//---------------------------------------------------------------------------------------------------------------
//
//  HAUD 2025.08.20
//
//  - XTS_TRANSPORT_LAYER
//
//  fb_StationBase
//  - abstract base class for XtsStation and XtsStationGearIn to extend
//  - anything goes..
//    - if you need a specialized station, use this so you can keep the control over the stations the same
//
//---------------------------------------------------------------------------------------------------------------
// This SOFTWARE is provided as an Example by THE PROVIDER "as is" and "with all faults." THE PROVIDER makes no 
// representations or warranties of any kind concerning the safety, suitability, lack of viruses, inaccuracies, 
// typographical errors, or other harmful components of this SOFTWARE. There are inherent dangers in the use of 
// any software, and you are solely responsible for determining whether this SOFTWARE is compatible with your 
// equipment and other software installed on your equipment. You are also solely responsible for the protection 
// of your equipment and backup of your data, and THE PROVIDER will not be liable for any damages you may suffer 
// in connection with using, modifying, or distributing this SOFTWARE.
//---------------------------------------------------------------------------------------------------------------
FUNCTION_BLOCK ABSTRACT fb_StationBase  IMPLEMENTS I_XtsTransport_Station
VAR
  _nStationId                 : UINT;  // why is Gamora?

  _eCheck                     : E_STATION_CHECK;  // additional output for Check()
  _eInitList                  : E_PROGRESS;       // linked list initialization progress
  _eFatalError                : E_STATION_STATE;

  // pointer to all stations
  _stCtrl                     : REFERENCE TO ARRAY[1..MAX_STATION]  OF ST_STATION_CTRL;   // are you talking to me?
  _stState                    : REFERENCE TO ARRAY[1..MAX_STATION]  OF ST_STATION_STATE;  // take the words right out of my mouth.

  // local copy of command
  _eCmd,
  _eCmdOld                    : E_STATION_CTRL; // this is a local shop for local people

  // through the looking class... yet near but so far
  // yes we use interfaces here
  _ItfStation                 : REFERENCE TO ARRAY[1..MAX_STATION]  OF I_Station_LinkedList;  // access to all stations lists
  _ItfMover                   : REFERENCE TO ARRAY[1..MAX_MOVER]    OF I_XtsTransport_Mover;  // access to mover methods

  // station related data
  _rMoverOffset               : REFERENCE TO ARRAY[1..MAX_STATION]  OF T_NEST_OFFSET;         // static offsets for station
  _stParameter                : REFERENCE TO ARRAY[1..MAX_STATION]  OF ST_STATION_PARAMETER;  // station parameter (where, how fast, how many stops)

  // mover axis ref for info
  _Mover                      : REFERENCE TO ARRAY[1..MAX_MOVER]    OF AXIS_REF;              // read from AXIS_REF

  // linked list result struct
  _stListEnter,
  _stListTarget,
  _stListDelete               : ST_STATION_LIST_RESULT;   // struct with result and ticket data

  _stMoverDataSend,
  _stMoverData                : ST_STATION_MOVER_DATA;    // mover ticket data

  _stInfeed,
  _stOutfeed                  : ST_MOVE_DATA;             // position and dynamic constraints of movement

  // work vars
  _Result                     : E_PROGRESS;               // it's a work in progress
  _eStateProgress             : E_PROGRESS;               // the fiddler on the roof (listen to him)

  _nNest,
  _nMoverDetected,
  _ix                         : UINT;

  _rModActPosFetch,
  _rPosInfeedMover            : LREAL;
  _bMatchMessageLevel         : BOOL := TRUE;   // TRUE --> Mover in Station commands have equal message level as station

  _stMsg                      : ST_Message;
  _eMessageLevel              : E_MessageType;
END_VAR

METHOD PROTECTED BitDel : WORD
VAR_INPUT
  inVal   : WORD;
  bitNo   : DINT;
END_VAR
VAR
  wConst : WORD := 1;
END_VAR
IF ( inVal AND SHL( wConst, TO_SINT(bitNo) MOD 16 ) ) > 0 THEN
  BitDel := inVal XOR (SHL( wConst,TO_SINT(bitNo) MOD 16 ));
ELSE
  BitDel := inVal;
END_IF
END_METHOD

METHOD PROTECTED BitGet : BOOL
VAR_INPUT
  inVal   : WORD;
  bitNo   : DINT;
END_VAR
VAR
  wConst : WORD := 1;
END_VAR
IF ( inVal AND SHL( wConst,TO_SINT(bitNo) MOD 16 ) ) > 0
THEN
  BitGet := TRUE;
ELSE
  BitGet := FALSE;
END_IF
END_METHOD

METHOD PROTECTED BitSet : WORD
VAR_INPUT
  inVal   : WORD;
  bitNo   : DINT;
END_VAR
VAR
  wConst  : WORD := 1;
END_VAR
BitSet := inVal OR SHL( wConst,TO_SINT(bitNo) MOD 16 );
END_METHOD

METHOD PROTECTED Check : BOOL
VAR_INPUT
END_VAR
                              // When the visionary dreams set hard and grey as flesh made into stone

IF NOT (_nStationId > 0) OR
       (_nStationId > MAX_STATION)
THEN
                              // You tore the statues to the ground crying - let my people go
  _eCheck                     := E_STATION_CHECK.STATION_ID_INVALID;
  RETURN;
END_IF

IF NOT __ISVALIDREF(_stCtrl)
THEN
                              // And now they're gone, all is gone
  _eCheck                     := E_STATION_CHECK.REFERENCE_CTRL_INVALID;
  RETURN;
END_IF

IF NOT __ISVALIDREF(_stState)
THEN
  _eCheck                     := E_STATION_CHECK.REFERENCE_STATE_INVALID;
  RETURN;
END_IF

IF NOT __ISVALIDREF(_ItfStation)
THEN
                              // They dance together upon the wall
                              // With nothing left to break the fall
  _eCheck                     := E_STATION_CHECK.REFERENCE_LIST_ITF_INVALID;
  RETURN;
END_IF

IF NOT __ISVALIDREF(_ItfMover)
THEN
  _eCheck                     := E_STATION_CHECK.REFERENCE_MOVER_ITF_INVALID;
  RETURN;
END_IF

IF NOT __ISVALIDREF(_rMoverOffset)
THEN
  _eCheck                     := E_STATION_CHECK.REFERENCE_MOVER_OFFSET_INVALID;
  RETURN;
END_IF

IF NOT __ISVALIDREF(_stParameter)
THEN
  _eCheck                     := E_STATION_CHECK.REFERENCE_PARAMETER_INVALID;
  RETURN;
END_IF

IF NOT __ISVALIDREF(_Mover)
THEN
  _eCheck                     := E_STATION_CHECK.REFERENCE_MOVER_AXIS_REF_INVALID;
  RETURN;
END_IF


_eCheck                       := E_STATION_CHECK.CHECK_DONE;
Check                         := TRUE;
END_METHOD

PROPERTY Ctrl : reference to ARRAY[1..MAX_STATION] OF ST_STATION_CTRL
SET
_stCtrl ref= Ctrl;
END_SET
END_PROPERTY

METHOD Cycle
VAR_INPUT
END_VAR
END_METHOD

METHOD Init : e_progress
VAR_INPUT
END_VAR
// check pointer and interface
IF NOT Check() THEN Init := e_progress.PROGRESS_ERROR; RETURN; END_IF

_stState[_nStationId].nMask       := 0;
_stState[_nStationId].nMoverId    := 0;

_eFatalError                      := E_STATION_STATE.STATION_ERROR_NULL;

_stState[_nStationId].State      := E_STATION_STATE.STATION_INIT;

IF _ItfStation[_nStationId].InitList()
THEN
  IF (_eMessageLevel = E_MessageType.eMessageVerbose)
  THEN
    _stMsg.eType                  := E_MessageType.eMessageVerbose;
    _stMsg.eSubdevice             := Stationstate;
    _stMsg.iErrorNumber           := 0;
    _stMsg.sText                  := concat('_ItfStation.InitList', ': ');
    _stMsg.sText                  := concat(_stMsg.sText, TO_STRING(E_PROGRESS.PROGRESS_DONE));
    //f_MessageSet(_stMsg);
  END_IF

  Init                            := E_PROGRESS.PROGRESS_DONE;

ELSE
    _stMsg.eType                  := E_MessageType.eMessageError;
    _stMsg.eSubdevice             := Stationstate;
    _stMsg.iErrorNumber           := 0;
    _stMsg.sText                  := concat('_ItfStation.InitList', ': ');
    _stMsg.sText                  := concat(_stMsg.sText, TO_STRING(E_PROGRESS.PROGRESS_ERROR));
    f_MessageSet(_stMsg);

  Init                            := e_progress.PROGRESS_ERROR;
END_IF
END_METHOD

PROPERTY ItfMover : reference to ARRAY[1..MAX_MOVER] OF I_XtsTransport_Mover
SET
_ItfMover ref= ItfMover;
END_SET
END_PROPERTY

PROPERTY ItfStations : reference to ARRAY[1..MAX_STATION] OF I_Station_LinkedList
SET
_ItfStation ref= ItfStations;
END_SET
END_PROPERTY

METHOD LogState
VAR_INPUT
  eType       : E_MessageType;
END_VAR
_stMsg.eType                := eType;
_stMsg.eSubdevice           := Stationstate;
_stMsg.iErrorNumber         := _stState[_nStationId].nMoverId;
_stMsg.sText                := TO_STRING(_stState[_nStationId].State);
f_MessageSet(_stMsg);
END_METHOD

PROPERTY MessageLevel : e_messagetype
SET
_eMessageLevel := MessageLevel;
END_SET
END_PROPERTY

METHOD MoveIn // prepares movement to PostStop[_nNest] in station
// build WorkPos from parameter, static station data and information on mover
_stInfeed.rPos            := _stParameter[_nStationId].rPosWait
                          +  _stParameter[_nStationId].rPosStop[_nNest]
                          +  _stMoverData.rOffset
                          +  _rMoverOffset[_nStationId][_stMoverData.nMoverId][_nNest];

_stInfeed.rVelo           := _stParameter[_nStationId].rVelo;
_stInfeed.rAcc            := _stParameter[_nStationId].rAccDec;
_stInfeed.rJerk           := _stParameter[_nStationId].rJerk;
_stInfeed.rGap            := _stParameter[_nStationId].rGap;
_stInfeed.rDistance       := _stParameter[_nStationId].rReleaseDistance;
_stInfeed.rDelta          := TargetWindow;

// init method
_ItfMover[_stState[_nStationId].nMoverId].MoveToPosCa(FALSE, _stInfeed);

// clear substate
_eStateProgress           := E_PROGRESS.PROGRESS_INIT;
END_METHOD

METHOD MoveOut // prepares mover data for sending to target station
// build data for sending mover to target station

// who am I sending?
_stMoverDataSend.nMoverId         := _stState[_nStationId].nMoverId;

// get optional information about nests to work
_stMoverDataSend.nMask            := _stCtrl[_nStationId].nMask;

// get optional offset
_stMoverDataSend.rOffset          := _stCtrl[_nStationId].rOffset;

// get target station
_stMoverDataSend.nTargetStation   := _stCtrl[_nStationId].nTargetStation;

// get position of target
_stOutfeed.rPos                   := _stParameter[_stMoverDataSend.nTargetStation].rPosWait;

IF (_stOutfeed.rPos - _Mover[_stMoverDataSend.nMoverId].NcToPlc.ModuloActPos < 0)
THEN
  // only forward, never back
  _stOutfeed.rPos             := _stOutfeed.rPos 
                              +  _ItfMover[_stMoverDataSend.nMoverId].RailLength;
END_IF

_stOutfeed.rVelo              := _stParameter[_nStationId].rVelo;
_stOutfeed.rAcc               := _stParameter[_nStationId].rAccDec;
_stOutfeed.rJerk              := _stParameter[_nStationId].rJerk;

IF (_stParameter[_nStationId].rGap > _stParameter[_stMoverDataSend.nTargetStation].rGap + 1.0)
THEN
  _stOutfeed.rGap             := _stParameter[_stMoverDataSend.nTargetStation].rGap;
ELSE
  _stOutfeed.rGap             := _stParameter[_nStationId].rGap;
END_IF

_stOutfeed.rDistance          := _stParameter[_nStationId].rReleaseDistance;

// init method for sending
_ItfMover[_stMoverDataSend.nMoverId].SendToModuloPosCa(FALSE, _stOutfeed);
END_METHOD

PROPERTY Mover : reference TO ARRAY[1..MAX_MOVER] OF AXIS_REF;
SET
_Mover ref= Mover;
END_SET
END_PROPERTY

PROPERTY MoverOffset : reference TO ARRAY[1..MAX_STATION]  OF T_NEST_OFFSET
SET
_rMoverOffset ref= MoverOffset;
END_SET
END_PROPERTY

PROPERTY State : reference to ARRAY[1..MAX_STATION] OF ST_STATION_STATE
SET
_stState ref= State;
END_SET
END_PROPERTY

PROPERTY StationId : uint
GET
StationId := _nStationId;
END_GET
SET
_nStationId := StationId;
END_SET
END_PROPERTY

PROPERTY StationParameter : reference TO ARRAY[1..MAX_STATION]  OF ST_STATION_PARAMETER
SET
_stParameter ref= StationParameter;
END_SET
END_PROPERTY

PROPERTY TargetWindow : lreal
GET
TargetWindow := SEL((_stInfeed.rDelta < 0.05), _stInfeed.rDelta, 0.1);
END_GET
SET
_stInfeed.rDelta := SEL((TargetWindow < 0.05), TargetWindow, 0.1);
END_SET
END_PROPERTY

END_FUNCTION_BLOCK

(* stored: Version 1.1.0.1, ProductVersion 3.1.4026.13
   POU fb_StationBase: Id {0b8dff22-a149-4a45-afd0-c2215976fd93}, SpecialFunc None
   Folder methods: Id {70829820-e56f-4eb2-b22e-8724574916a3}
   Folder properties: Id {a4e8a5c0-089d-4736-a684-5b0f4b556517}
   Method BitDel: Id {0be77e49-7392-4c3c-a864-49cf6caf7308}
   Method BitGet: Id {d8ce1ab4-8924-4075-8c23-01c3fb056560}
   Method BitSet: Id {93ad0b2a-1657-4728-8c02-324c1b2a5b28}
   Method Check: Id {e1ef4bef-70bf-4332-81e2-483f8385e36d}
   Property Ctrl: Id {9c1d9a11-da8a-4ba2-8182-211097542342}
   Set Set: Id {a26c4996-5a5d-42c0-896e-271173b65645}
   Method Cycle: Id {79caa820-ee26-4207-a9dd-9effc321454e}
   Method Init: Id {a797a9db-4c0e-424f-8156-620d128fdf6c}
   Property ItfMover: Id {71937b15-91ca-4496-bdc4-b61532cb5c65}
   Set Set: Id {45f74677-7c1c-4f34-bbf4-37f8ad9a6065}
   Property ItfStations: Id {f5e91a53-1425-4cbb-bc1f-49b9b9b76cc7}
   Set Set: Id {2ec3c429-b30b-47c3-b5d8-ba92b6a18168}
   Method LogState: Id {b099bac2-7924-43f7-b859-60dcfdd23a11}
   Property MessageLevel: Id {19cf9e40-f4f2-4a59-b342-a999c05b9027}
   Set Set: Id {06a23d40-fab1-4a04-8d5f-bd8a56548582}
   Method MoveIn: Id {c0f47d1b-64fd-4c72-a6ef-0fbc75011c35}
   Method MoveOut: Id {cc449cf5-a2c5-42b1-8e22-522047389dd2}
   Property Mover: Id {e82910a4-d871-4e5e-b77c-c01f33e3b55d}
   Set Set: Id {44ec8ec6-bdc8-49bb-b3f3-a1d3bd8ab268}
   Property MoverOffset: Id {4a4324a4-0c99-4891-9585-78144eecb105}
   Set Set: Id {afb8fc34-701f-4fcb-bc3a-f0cae488d17a}
   Property State: Id {ea1d69aa-9e7b-43c0-803d-987ed4934b15}
   Set Set: Id {7e8ecc2e-d8ce-493a-a8c4-0138cc2cb66a}
   Property StationId: Id {f440e647-2b56-47f6-9e54-30e69375a6c1}
   Get Get: Id {7f95c3ff-d25a-49a2-83f5-6a8f8da9f016}
   Set Set: Id {0746dd45-9ceb-4162-a875-ac226e6b452a}
   Property StationParameter: Id {07bf2b08-2b73-4810-bdf6-9da9a74a1847}
   Set Set: Id {cd69203e-8d66-4e00-bdb1-edbcf15b620c}
   Property TargetWindow: Id {392ae526-9be1-4234-afa2-c2662dd1fbbd}
   Get Get: Id {79f50164-d3cd-4bf2-a579-3ab0b195682d}
   Set Set: Id {69dea1a4-0e95-43a8-b90d-b04f5beda7b5} *)
